FUNCTION_BLOCK GET_1D_COORD (* Set coordinates for 1D movement destination *)
  (* Standard: 61499-2 *)
  (* Version 1.0, 23-03-12, GASR, Universidade do Estado de Santa Catarina *)
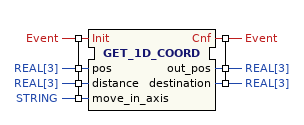
  EVENT_INPUT
    Init WITH pos, distance, move_in_axis; (* Initialization Request *)
  END_EVENT
  EVENT_OUTPUT
    Cnf WITH out_pos, destination; (* Execution confirmed *)
  END_EVENT
  VAR_INPUT
    pos : ARRAY [0..2] OF REAL; (* Machine position *)
    distance : ARRAY [0..2] OF REAL; (* Distance *)
    move_in_axis : STRING; (* x, y or z axis? *)
  END_VAR
  VAR_OUTPUT
    out_pos : ARRAY [0..2] OF REAL;
    destination : ARRAY [0..2] OF REAL;
  END_VAR
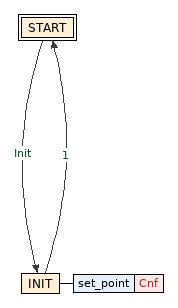
  EC_STATES
    START; (* Initial state *)
    INIT : set_point -> Cnf; (* Algorithm execution *)
  END_STATES
  EC_TRANSITIONS
    START TO INIT := Init;
    INIT TO START := 1;
  END_TRANSITIONS
  ALGORITHM set_point IN Lua:
out_pos[1]     = pos[1]
out_pos[2]     = pos[2]
out_pos[3]     = pos[3]
destination[1] = pos[1]
destination[2] = pos[2]
destination[3] = pos[3]
if( move_in_axis == 'x' ) then
	destination[1] = distance[1]
elseif( move_in_axis == 'y' ) then
	destination[2] = distance[2]
elseif( move_in_axis == 'z' ) then
	destination[3] = distance[3]
end
  END_ALGORITHM
END_FUNCTION_BLOCK
